{attribute 'no_explicit_call' := 'Gate is a CLASS and must be accessed using methods or properties'}
FUNCTION_BLOCK Gate IMPLEMENTS I_OpenCommand, I_CloseCommand
VAR
	open						AT %Q*: BOOL;
	close						AT %Q*: BOOL;
	_isOpen						AT %I*: BOOL;
	_isClosed					AT %I*: BOOL;
END_VAR


// The body of a class must not be used for code.  
// Cyclic code should be called from a method if needed.

METHOD Close
open := FALSE;
close := NOT isClosed; // Close until closed
END_METHOD

PROPERTY IsClosed : BOOL
GET
IsClosed := _isClosed;
END_GET
END_PROPERTY

PROPERTY IsOpen : BOOL
GET
IsOpen := _isOpen;
END_GET
END_PROPERTY

METHOD Open
close := FALSE;
open := NOT isOpen; // Open until opened
END_METHOD

END_FUNCTION_BLOCK

(* stored: Version 1.1.0.1, ProductVersion 3.1.4024.11
   POU Gate: Id {8a1d58b5-97e9-41da-a416-67ec0319fefe}, SpecialFunc None
   Method Close: Id {666587c5-fa1b-4054-884f-aaf313e6576b}
   Property IsClosed: Id {4d8ef7ea-6f63-4e42-bb3b-6033d89c734a}
   Get Get: Id {1ce93ebe-e313-4e65-a214-c29b53054926}
   Property IsOpen: Id {dfca3071-e9a1-406c-b6af-4d1734797639}
   Get Get: Id {eb3e1315-78cd-4510-a440-b04891e16339}
   Method Open: Id {a14af5e6-4339-4ef8-a520-e610eb7c0e84} *)
